PROGRAM P_CoatingProtections
VAR
    	fbStripProtMR1L0 : FB_MirrorTwoCoatingProtection := (
            sDevName := 'MR1L0',
            nUpperCoatingBoundary := 13300000,
            nUpperCoatingBitmask := 2#0000_0000_0000_0000_1111_1111_1111_1100, // Exclusion range 0,1 AND 14,90
            sUpperCoatingType := 'B4C',
            nLowerCoatingBoundary := 11800000,
            nLowerCoatingBitMask := 2#0011_1111_1111_1111_1110_0000_0000_0000, //exclusion range 0,12 AND 27???,90
            sLowerCoatingType := 'B4C/Ni');

    	fbStripProtMR2L0 : FB_MirrorTwoCoatingProtection := (
            sDevName := 'MR2L0',
            nUpperCoatingBoundary := 14300000,
            nUpperCoatingBitmask := 2#0000_0000_0000_0000_1111_1111_1111_1100, // Exclusion range 0,1 AND 14,90
            sUpperCoatingType := 'Ni',
            nLowerCoatingBoundary := 12800000,
            nLowerCoatingBitMask :=  2#0011_1111_1111_1111_1110_0000_0000_0000, //exclusion range 0,12 AND 27???,90
            sLowerCoatingType := 'B4C');
END_VAR

fbStripProtMR1L0(
    nCurrentEncoderCount := MAIN.nEncCntYupM1L0,
    neVRange := PMPS.PMPS_GVL.stCurrentBeamParameters.neVRange,
    FFO := GVL_PMPS.g_FastFaultOutput1);
    
fbStripProtMR2L0(
    nCurrentEncoderCount := MAIN.nEncCntYupM2L0,
    neVRange := PMPS.PMPS_GVL.stCurrentBeamParameters.neVRange,
    FFO := GVL_PMPS.g_FastFaultOutput1);

END_PROGRAM

(* stored: Version 1.1.0.1, ProductVersion 3.1.4022.18
   POU P_CoatingProtections: Id {3eac67bd-ceb1-46f6-9fb2-5e3c0612d4cd}, SpecialFunc None *)
